// TIA Portal V16 export
// export: Created 2021-11-12T13:32:29.9953975Z, ExportSetting WithDefaults, DisplayName Totally Integrated Automation Portal, DisplayVersion V16 Update 3, DisplayName TIA Portal Version Control Interface, DisplayVersion V16 Update 2, DisplayName TIA Portal Openness, DisplayVersion V16 Update 3, DisplayName SINAMICS Startdrive Advanced, DisplayVersion V16 Update 5, DisplayName SINAMICS Startdrive G130, G150, S120, S150, SINAMICS MV, S210, DisplayVersion V16 Update 5, DisplayName SINAMICS Startdrive G110M, G120, G120C, G120D, G120P, G115D, DisplayVersion V16 Update 5, DisplayName STEP 7 Professional, DisplayVersion V16 Update 3, DisplayName STEP 7 Safety, DisplayVersion V16, DisplayName WinCC UA Professional, DisplayVersion V16 Update 3
DATA_BLOCK "STATUS_1R3"   // DB135
{ S7_Optimized_Access := 'TRUE' }
VERSION : 0.1
// stored: AutoNumber true, DBAccessibleFromOPCUA true, IsOnlyStoredInLoadMemory false, IsRetainMemResEnabled false, IsWriteProtectedInAS false, MemoryReserve 100
   VAR
      xxxxx___BinarySensors___xxxxx : Byte;
      "CL01-BG01_4" : Bool;   // Robot 1R3 Gripper on table 1
      "CL02-BG01_4" : Bool;   // Robot 1R3 Gripper on table 2
      "RO01-BG10_2" : Bool;   // Robot 1R3 senzor piston lubrication printed / Robot 1R3 senzor pístu mazivo vytlačeno
      xxxxx___BinaryOthers___xxxxx : Byte;
      PwrOK : Bool;
      "100+UF01-SF02_12" : Bool;   // Robot 1R3, 1R4 immediate stop
      "000+UH10-SF26_12" : Bool;   // Okamžitý stop Robot 1R3, 1R4
      RobotNotUsed : Bool;   // Robot is not used
      xxxxx___AnalogueSensors___xxxxx : Byte;
      xxxxx___Drives___xxxxx : Byte;
      RO01 : Struct   // Robot
         Main : "UDT_Status_main";
         Specific : "UDT_RobotABB_Status_specific";
         Error : "UDT_Error01";
      END_STRUCT;
      RC01 : Struct   // Controller
         Main : "UDT_Status_main";
         Specific : "UDT_DriveRobotABB_Status_specific";
         Error : "UDT_Error01";
      END_STRUCT;
      Gripper : Struct   // Gripper
         Main : "UDT_Status_main";
         Specific : "UDT_RobotGripper_Status_specific";
         Error : "UDT_Error10";
      END_STRUCT;
      xxxxx___Others___xxxxx : Byte;
      Interlocks { S7_SetPoint := 'True'} : "UDT_RobotABB_Interlock";
      ZoneRelease { S7_SetPoint := 'True'} : "UDT_RobotABB_ZoneReleaseToRobot";
      "Counter" { S7_SetPoint := 'True'} : Int;   // Number of parts in gripper
      Sequence : Struct
         Main : "UDT_Status_main";
         Specific { S7_SetPoint := 'True'} : "UDT_Sequence_Status_Specific";
         Error { S7_SetPoint := 'True'} : "UDT_Error01";
      END_STRUCT;
      xxxxx___MaterialFlow___xxxxx_1 { S7_SetPoint := 'True'} : Byte;
   END_VAR
   VAR RETAIN
      MatCard : Array[1..4, 1..2] of "UDT_MatCard";   // Material card [Line - shorter side, Row - longer side]
   END_VAR
   VAR
      xxxxx___Alarms___xxxxx : Byte;
      RO01_Timeout : Struct   // Robot job active for too long / Job robota aktivní příliš dlhou dobu.
         Main { S7_SetPoint := 'True'} : "UDT_Status_main";
         Specific { S7_SetPoint := 'True'} : "UDT_DI_Mon_Status_specific";
         Error { S7_SetPoint := 'True'} : "UDT_Error01";
      END_STRUCT;
      CL01_BG01 : Struct   // Gripper on upper table / Chapadlo na horním odkládacím stolku.
         Main { S7_SetPoint := 'True'} : "UDT_Status_main";
         Specific { S7_SetPoint := 'True'} : "UDT_DI_Mon_Status_specific";
         Error { S7_SetPoint := 'True'} : "UDT_Error01";
      END_STRUCT;
      CL01_BG02 : Struct   // Gripper on lower table / Chapadlo na dolním odkládacím stolku.
         Main { S7_SetPoint := 'True'} : "UDT_Status_main";
         Specific { S7_SetPoint := 'True'} : "UDT_DI_Mon_Status_specific";
         Error { S7_SetPoint := 'True'} : "UDT_Error01";
      END_STRUCT;
      ES : Struct   // E-stop
         Main { S7_SetPoint := 'True'} : "UDT_Status_main";
         Specific { S7_SetPoint := 'True'} : "UDT_DI_Mon_Status_specific";
         Error { S7_SetPoint := 'True'} : "UDT_Error01";
      END_STRUCT;
      "RO01-BG10" : Struct   // Robot 1R3 senzor piston lubrication not printed / Robot 1R3 senzor pístu mazivo nevytlačeno
         Main { S7_SetPoint := 'True'} : "UDT_Status_main";
         Specific { S7_SetPoint := 'True'} : "UDT_DI_Mon_Status_specific";
         Error { S7_SetPoint := 'True'} : "UDT_Error01";
      END_STRUCT;
   END_VAR
BEGIN
END_DATA_BLOCK
